// TIA Portal V17 export
// export: Created 2025-03-10T12:16:31.661415Z, ExportSetting WithDefaults, DisplayName Totally Integrated Automation Portal, DisplayVersion V17 Update 8, DisplayName TIA Portal Openness, DisplayVersion V17 Update 8, DisplayName TIA Portal Version Control Interface, DisplayVersion V17, DisplayName SINAMICS Startdrive Advanced, DisplayVersion V17 SP2, DisplayName SINAMICS Startdrive G110M, G120, G120C, G120D, G120P, G115D, DisplayVersion V17 SP2, DisplayName SINAMICS Startdrive G130, G150, S120, S150, SINAMICS MV, S210, DisplayVersion V17 SP2, DisplayName STEP 7 Professional, DisplayVersion V17 Update 8, DisplayName SINUMERIK ONE STEP 7 Toolbox, DisplayVersion V17 Update 12, DisplayName SINUMERIK 840D sl STEP 7 Toolbox, DisplayVersion V17 Update 12, DisplayName STEP 7 Safety, DisplayVersion V17 Update 6, DisplayName WinCC Advanced, DisplayVersion V17 Update 8
DATA_BLOCK "DB1714_UNIT_01_STA_4_ASPIRATION_VALVE"   // DB1714
{ DB_Accessible_From_OPC_UA := 'FALSE' }
VERSION : 0.1
// stored: AutoNumber false, DBAccessibleFromOPCUA false, DBAccessibleFromWebserver true, InstanceOfName FB1702_ASPIRATION_VALVE, InstanceOfType FB
"FB1702_ASPIRATION_VALVE"
   // VAR_INPUT
   //    OPTIONS_0 : Byte;
   //    FLOW_PRESENT_INPUT_1 : Bool;
   //    FLOW_PRESENT_INPUT_2 : Bool;
   //    SWITCH_ON_CONDITIONS : Bool;
   //    SWITCH_OFF_CONDITIONS : Bool;
   //    HMI_LINE_REQUEST : Bool;
   //    SWITCH_ON_AUTO_REQUEST : Bool;
   //    SWITCH_OFF_AUTO_REQUEST : Bool;
   //    SWITCH_OFF_GLOBAL_REQUEST : Bool;
   //    UNIT_ALARM : UInt;
   //    STATION_ALARM : UInt;
   // END_VAR
   // VAR_OUTPUT
   //    SWITCHED_ON : Bool;
   //    SWITCHED_OFF : Bool;
   //    SIMULTANEITY_ALARM : Bool;
   //    TIME_EXCEEDED_ALARM : Bool;
   //    SWITCH_ON_ALARM : Bool;
   //    SWITCH_OFF_ALARM : Bool;
   //    HMI_MOTION_EXECUTABILITY_LEFT : Bool;
   //    HMI_MOTION_EXECUTABILITY_RIGHT : Bool;
   //    HMI_MOTION_END_POS_LEFT : Bool;
   //    HMI_MOTION_END_POS_RIGHT : Bool;
   //    HMI_MOTION_ACTIVE_LEFT : Bool;
   //    HMI_MOTION_ACTIVE_RIGHT : Bool;
   //    SWITCH_ON : Bool;
   //    SWITCH_OFF : Bool;
   // END_VAR
   // VAR RETAIN
   //    CYL { S7_SetPoint := 'True'} : "ASPIRATION";
   //    TIMER_SWITCHED_ON { S7_SetPoint := 'True'} : TON_TIME;
   //    TIMER_SWITCHED_OFF { S7_SetPoint := 'True'} : TON_TIME;
   //    TIMER_SIMULTANEITY { S7_SetPoint := 'True'} : TON_TIME;
   //    TIMER_TIME_EXCEEDED { S7_SetPoint := 'True'} : TON_TIME;
   //    PULSE { S7_SetPoint := 'True'} : Bool;
   // END_VAR
BEGIN
END_DATA_BLOCK
